// TIA Portal V16 export
// export: Created 2021-04-11T09:51:25.5675002Z, ExportSetting WithDefaults, DisplayName Totally Integrated Automation Portal, DisplayVersion V16, DisplayName TIA Portal Version Control Interface, DisplayVersion V16, DisplayName TIA Portal Openness, DisplayVersion V16, DisplayName STEP 7 Professional, DisplayVersion V16, DisplayName STEP 7 Safety, DisplayVersion V16, DisplayName WinCC Unified SCADA Engineering System, DisplayVersion V16
FUNCTION "DBtoIO" : Void   // FC2, LAD
{ S7_Optimized_Access := 'TRUE' }
VERSION : 0.1
// stored: AutoNumber true, IsIECCheckEnabled false, SetENOAutomatically false, UDAEnableTagReadback false
BEGIN

REGION Network 1: Конвейер1 - вперед
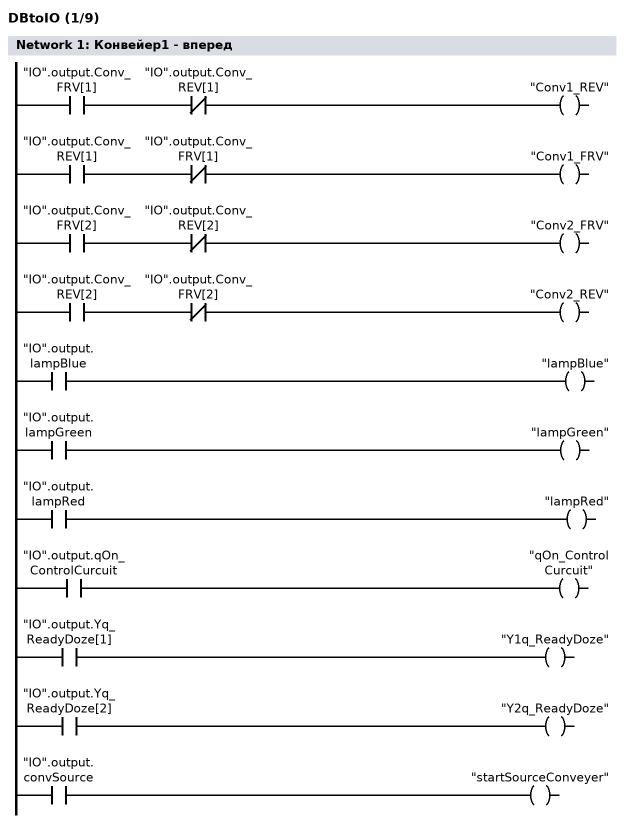
   RUNG wire#powerrail
      Contact( "IO".output.Conv_FRV[1] )
      I_Contact( "IO".output.Conv_REV[1] )
      Coil( "Conv1_REV" )
   END_RUNG
   RUNG wire#powerrail
      Contact( "IO".output.Conv_REV[1] )
      I_Contact( "IO".output.Conv_FRV[1] )
      Coil( "Conv1_FRV" )
   END_RUNG
   RUNG wire#powerrail
      Contact( "IO".output.Conv_FRV[2] )
      I_Contact( "IO".output.Conv_REV[2] )
      Coil( "Conv2_FRV" )
   END_RUNG
   RUNG wire#powerrail
      Contact( "IO".output.Conv_REV[2] )
      I_Contact( "IO".output.Conv_FRV[2] )
      Coil( "Conv2_REV" )
   END_RUNG
   RUNG wire#powerrail
      Contact( "IO".output.lampBlue )
      Coil( "lampBlue" )
   END_RUNG
   RUNG wire#powerrail
      Contact( "IO".output.lampGreen )
      Coil( "lampGreen" )
   END_RUNG
   RUNG wire#powerrail
      Contact( "IO".output.lampRed )
      Coil( "lampRed" )
   END_RUNG
   RUNG wire#powerrail
      Contact( "IO".output.qOn_ControlCurcuit )
      Coil( "qOn_ControlCurcuit" )
   END_RUNG
   RUNG wire#powerrail
      Contact( "IO".output.Yq_ReadyDoze[1] )
      Coil( "Y1q_ReadyDoze" )
   END_RUNG
   RUNG wire#powerrail
      Contact( "IO".output.Yq_ReadyDoze[2] )
      Coil( "Y2q_ReadyDoze" )
   END_RUNG
   RUNG wire#powerrail
      Contact( "IO".output.convSource )
      Coil( "startSourceConveyer" )
   END_RUNG
   // the same network as SCL:
   "Conv1_REV" := "IO".output.Conv_FRV[1] AND NOT "IO".output.Conv_REV[1];
   "Conv1_FRV" := "IO".output.Conv_REV[1] AND NOT "IO".output.Conv_FRV[1];
   "Conv2_FRV" := "IO".output.Conv_FRV[2] AND NOT "IO".output.Conv_REV[2];
   "Conv2_REV" := "IO".output.Conv_REV[2] AND NOT "IO".output.Conv_FRV[2];
   "lampBlue" := "IO".output.lampBlue;
   "lampGreen" := "IO".output.lampGreen;
   "lampRed" := "IO".output.lampRed;
   "qOn_ControlCurcuit" := "IO".output.qOn_ControlCurcuit;
   "Y1q_ReadyDoze" := "IO".output.Yq_ReadyDoze[1];
   "Y2q_ReadyDoze" := "IO".output.Yq_ReadyDoze[2];
   "startSourceConveyer" := "IO".output.convSource;
END_REGION

REGION Network 2: Управление открыванием лопаток - из массива в катушки
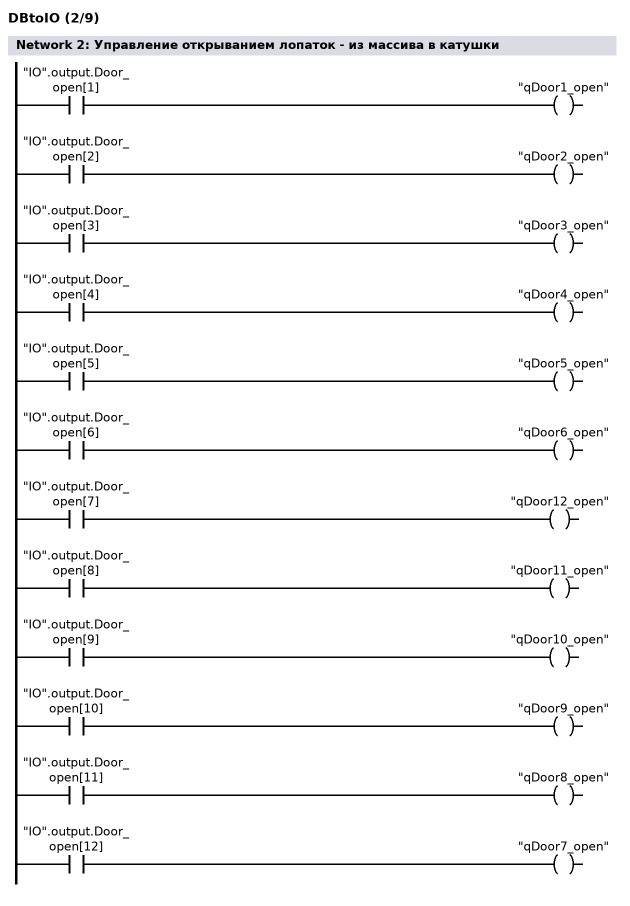
   RUNG wire#powerrail
      Contact( "IO".output.Door_open[1] )
      Coil( "qDoor1_open" )
   END_RUNG
   RUNG wire#powerrail
      Contact( "IO".output.Door_open[2] )
      Coil( "qDoor2_open" )
   END_RUNG
   RUNG wire#powerrail
      Contact( "IO".output.Door_open[3] )
      Coil( "qDoor3_open" )
   END_RUNG
   RUNG wire#powerrail
      Contact( "IO".output.Door_open[4] )
      Coil( "qDoor4_open" )
   END_RUNG
   RUNG wire#powerrail
      Contact( "IO".output.Door_open[5] )
      Coil( "qDoor5_open" )
   END_RUNG
   RUNG wire#powerrail
      Contact( "IO".output.Door_open[6] )
      Coil( "qDoor6_open" )
   END_RUNG
   RUNG wire#powerrail
      Contact( "IO".output.Door_open[7] )
      Coil( "qDoor12_open" )
   END_RUNG
   RUNG wire#powerrail
      Contact( "IO".output.Door_open[8] )
      Coil( "qDoor11_open" )
   END_RUNG
   RUNG wire#powerrail
      Contact( "IO".output.Door_open[9] )
      Coil( "qDoor10_open" )
   END_RUNG
   RUNG wire#powerrail
      Contact( "IO".output.Door_open[10] )
      Coil( "qDoor9_open" )
   END_RUNG
   RUNG wire#powerrail
      Contact( "IO".output.Door_open[11] )
      Coil( "qDoor8_open" )
   END_RUNG
   RUNG wire#powerrail
      Contact( "IO".output.Door_open[12] )
      Coil( "qDoor7_open" )
   END_RUNG
   // the same network as SCL:
   "qDoor1_open" := "IO".output.Door_open[1];
   "qDoor2_open" := "IO".output.Door_open[2];
   "qDoor3_open" := "IO".output.Door_open[3];
   "qDoor4_open" := "IO".output.Door_open[4];
   "qDoor5_open" := "IO".output.Door_open[5];
   "qDoor6_open" := "IO".output.Door_open[6];
   "qDoor12_open" := "IO".output.Door_open[7];
   "qDoor11_open" := "IO".output.Door_open[8];
   "qDoor10_open" := "IO".output.Door_open[9];
   "qDoor9_open" := "IO".output.Door_open[10];
   "qDoor8_open" := "IO".output.Door_open[11];
   "qDoor7_open" := "IO".output.Door_open[12];
END_REGION

REGION Network 3: Управление лопатки закрыть - из массива в катушки
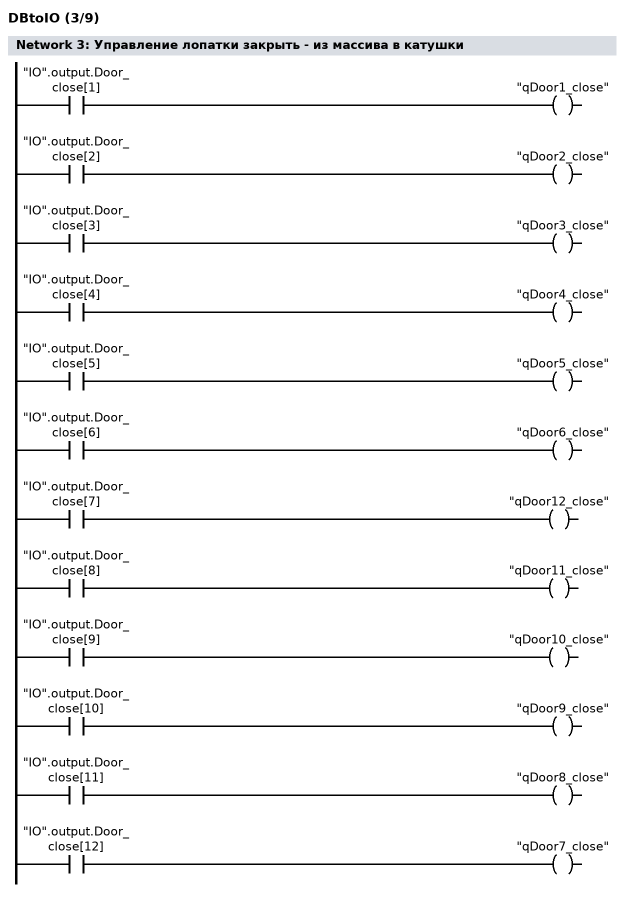
   RUNG wire#powerrail
      Contact( "IO".output.Door_close[1] )
      Coil( "qDoor1_close" )
   END_RUNG
   RUNG wire#powerrail
      Contact( "IO".output.Door_close[2] )
      Coil( "qDoor2_close" )
   END_RUNG
   RUNG wire#powerrail
      Contact( "IO".output.Door_close[3] )
      Coil( "qDoor3_close" )
   END_RUNG
   RUNG wire#powerrail
      Contact( "IO".output.Door_close[4] )
      Coil( "qDoor4_close" )
   END_RUNG
   RUNG wire#powerrail
      Contact( "IO".output.Door_close[5] )
      Coil( "qDoor5_close" )
   END_RUNG
   RUNG wire#powerrail
      Contact( "IO".output.Door_close[6] )
      Coil( "qDoor6_close" )
   END_RUNG
   RUNG wire#powerrail
      Contact( "IO".output.Door_close[7] )
      Coil( "qDoor12_close" )
   END_RUNG
   RUNG wire#powerrail
      Contact( "IO".output.Door_close[8] )
      Coil( "qDoor11_close" )
   END_RUNG
   RUNG wire#powerrail
      Contact( "IO".output.Door_close[9] )
      Coil( "qDoor10_close" )
   END_RUNG
   RUNG wire#powerrail
      Contact( "IO".output.Door_close[10] )
      Coil( "qDoor9_close" )
   END_RUNG
   RUNG wire#powerrail
      Contact( "IO".output.Door_close[11] )
      Coil( "qDoor8_close" )
   END_RUNG
   RUNG wire#powerrail
      Contact( "IO".output.Door_close[12] )
      Coil( "qDoor7_close" )
   END_RUNG
   // the same network as SCL:
   "qDoor1_close" := "IO".output.Door_close[1];
   "qDoor2_close" := "IO".output.Door_close[2];
   "qDoor3_close" := "IO".output.Door_close[3];
   "qDoor4_close" := "IO".output.Door_close[4];
   "qDoor5_close" := "IO".output.Door_close[5];
   "qDoor6_close" := "IO".output.Door_close[6];
   "qDoor12_close" := "IO".output.Door_close[7];
   "qDoor11_close" := "IO".output.Door_close[8];
   "qDoor10_close" := "IO".output.Door_close[9];
   "qDoor9_close" := "IO".output.Door_close[10];
   "qDoor8_close" := "IO".output.Door_close[11];
   "qDoor7_close" := "IO".output.Door_close[12];
END_REGION

REGION Network 4: Управление открыванием левым бункером - из массива в катушки
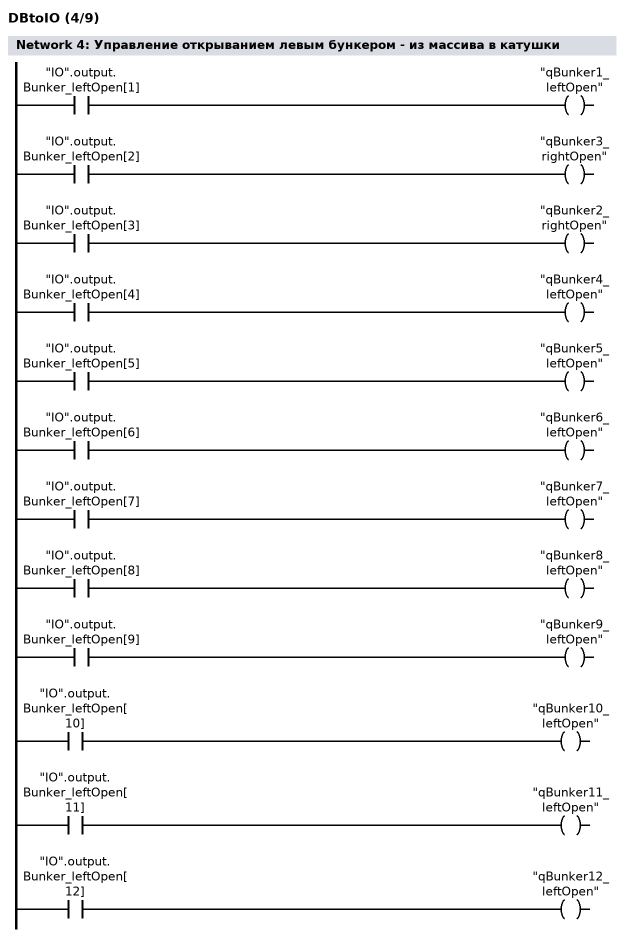
   RUNG wire#powerrail
      Contact( "IO".output.Bunker_leftOpen[1] )
      Coil( "qBunker1_leftOpen" )
   END_RUNG
   RUNG wire#powerrail
      Contact( "IO".output.Bunker_leftOpen[2] )
      Coil( "qBunker3_rightOpen" )
   END_RUNG
   RUNG wire#powerrail
      Contact( "IO".output.Bunker_leftOpen[3] )
      Coil( "qBunker2_rightOpen" )
   END_RUNG
   RUNG wire#powerrail
      Contact( "IO".output.Bunker_leftOpen[4] )
      Coil( "qBunker4_leftOpen" )
   END_RUNG
   RUNG wire#powerrail
      Contact( "IO".output.Bunker_leftOpen[5] )
      Coil( "qBunker5_leftOpen" )
   END_RUNG
   RUNG wire#powerrail
      Contact( "IO".output.Bunker_leftOpen[6] )
      Coil( "qBunker6_leftOpen" )
   END_RUNG
   RUNG wire#powerrail
      Contact( "IO".output.Bunker_leftOpen[7] )
      Coil( "qBunker7_leftOpen" )
   END_RUNG
   RUNG wire#powerrail
      Contact( "IO".output.Bunker_leftOpen[8] )
      Coil( "qBunker8_leftOpen" )
   END_RUNG
   RUNG wire#powerrail
      Contact( "IO".output.Bunker_leftOpen[9] )
      Coil( "qBunker9_leftOpen" )
   END_RUNG
   RUNG wire#powerrail
      Contact( "IO".output.Bunker_leftOpen[10] )
      Coil( "qBunker10_leftOpen" )
   END_RUNG
   RUNG wire#powerrail
      Contact( "IO".output.Bunker_leftOpen[11] )
      Coil( "qBunker11_leftOpen" )
   END_RUNG
   RUNG wire#powerrail
      Contact( "IO".output.Bunker_leftOpen[12] )
      Coil( "qBunker12_leftOpen" )
   END_RUNG
   // the same network as SCL:
   "qBunker1_leftOpen" := "IO".output.Bunker_leftOpen[1];
   "qBunker3_rightOpen" := "IO".output.Bunker_leftOpen[2];
   "qBunker2_rightOpen" := "IO".output.Bunker_leftOpen[3];
   "qBunker4_leftOpen" := "IO".output.Bunker_leftOpen[4];
   "qBunker5_leftOpen" := "IO".output.Bunker_leftOpen[5];
   "qBunker6_leftOpen" := "IO".output.Bunker_leftOpen[6];
   "qBunker7_leftOpen" := "IO".output.Bunker_leftOpen[7];
   "qBunker8_leftOpen" := "IO".output.Bunker_leftOpen[8];
   "qBunker9_leftOpen" := "IO".output.Bunker_leftOpen[9];
   "qBunker10_leftOpen" := "IO".output.Bunker_leftOpen[10];
   "qBunker11_leftOpen" := "IO".output.Bunker_leftOpen[11];
   "qBunker12_leftOpen" := "IO".output.Bunker_leftOpen[12];
END_REGION

REGION Network 5: Управление закрытием левым бункером - из массива в катушки
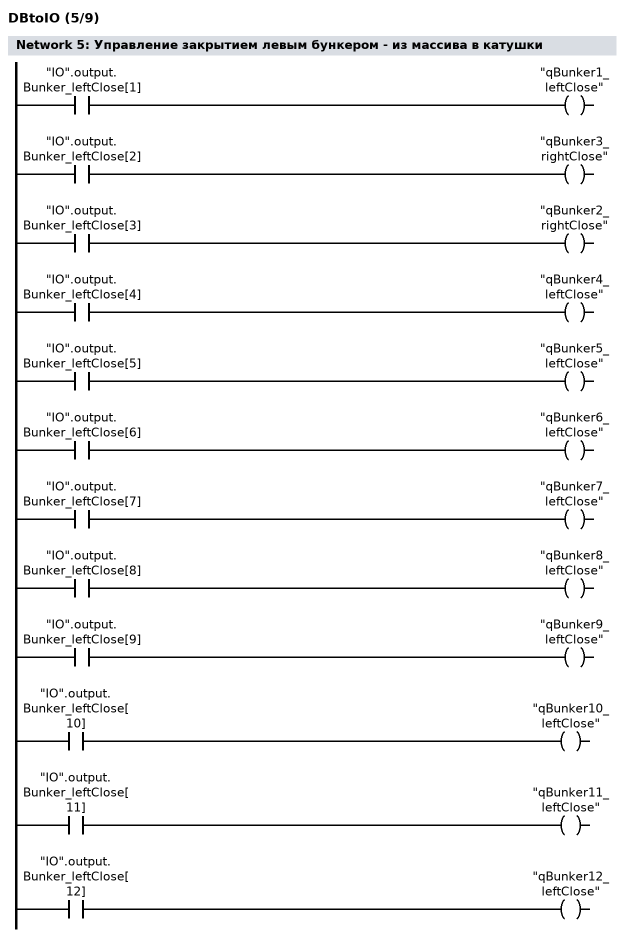
   RUNG wire#powerrail
      Contact( "IO".output.Bunker_leftClose[1] )
      Coil( "qBunker1_leftClose" )
   END_RUNG
   RUNG wire#powerrail
      Contact( "IO".output.Bunker_leftClose[2] )
      Coil( "qBunker3_rightClose" )
   END_RUNG
   RUNG wire#powerrail
      Contact( "IO".output.Bunker_leftClose[3] )
      Coil( "qBunker2_rightClose" )
   END_RUNG
   RUNG wire#powerrail
      Contact( "IO".output.Bunker_leftClose[4] )
      Coil( "qBunker4_leftClose" )
   END_RUNG
   RUNG wire#powerrail
      Contact( "IO".output.Bunker_leftClose[5] )
      Coil( "qBunker5_leftClose" )
   END_RUNG
   RUNG wire#powerrail
      Contact( "IO".output.Bunker_leftClose[6] )
      Coil( "qBunker6_leftClose" )
   END_RUNG
   RUNG wire#powerrail
      Contact( "IO".output.Bunker_leftClose[7] )
      Coil( "qBunker7_leftClose" )
   END_RUNG
   RUNG wire#powerrail
      Contact( "IO".output.Bunker_leftClose[8] )
      Coil( "qBunker8_leftClose" )
   END_RUNG
   RUNG wire#powerrail
      Contact( "IO".output.Bunker_leftClose[9] )
      Coil( "qBunker9_leftClose" )
   END_RUNG
   RUNG wire#powerrail
      Contact( "IO".output.Bunker_leftClose[10] )
      Coil( "qBunker10_leftClose" )
   END_RUNG
   RUNG wire#powerrail
      Contact( "IO".output.Bunker_leftClose[11] )
      Coil( "qBunker11_leftClose" )
   END_RUNG
   RUNG wire#powerrail
      Contact( "IO".output.Bunker_leftClose[12] )
      Coil( "qBunker12_leftClose" )
   END_RUNG
   // the same network as SCL:
   "qBunker1_leftClose" := "IO".output.Bunker_leftClose[1];
   "qBunker3_rightClose" := "IO".output.Bunker_leftClose[2];
   "qBunker2_rightClose" := "IO".output.Bunker_leftClose[3];
   "qBunker4_leftClose" := "IO".output.Bunker_leftClose[4];
   "qBunker5_leftClose" := "IO".output.Bunker_leftClose[5];
   "qBunker6_leftClose" := "IO".output.Bunker_leftClose[6];
   "qBunker7_leftClose" := "IO".output.Bunker_leftClose[7];
   "qBunker8_leftClose" := "IO".output.Bunker_leftClose[8];
   "qBunker9_leftClose" := "IO".output.Bunker_leftClose[9];
   "qBunker10_leftClose" := "IO".output.Bunker_leftClose[10];
   "qBunker11_leftClose" := "IO".output.Bunker_leftClose[11];
   "qBunker12_leftClose" := "IO".output.Bunker_leftClose[12];
END_REGION

REGION Network 6: Управление открыванием правого бункера - из массива в катушки
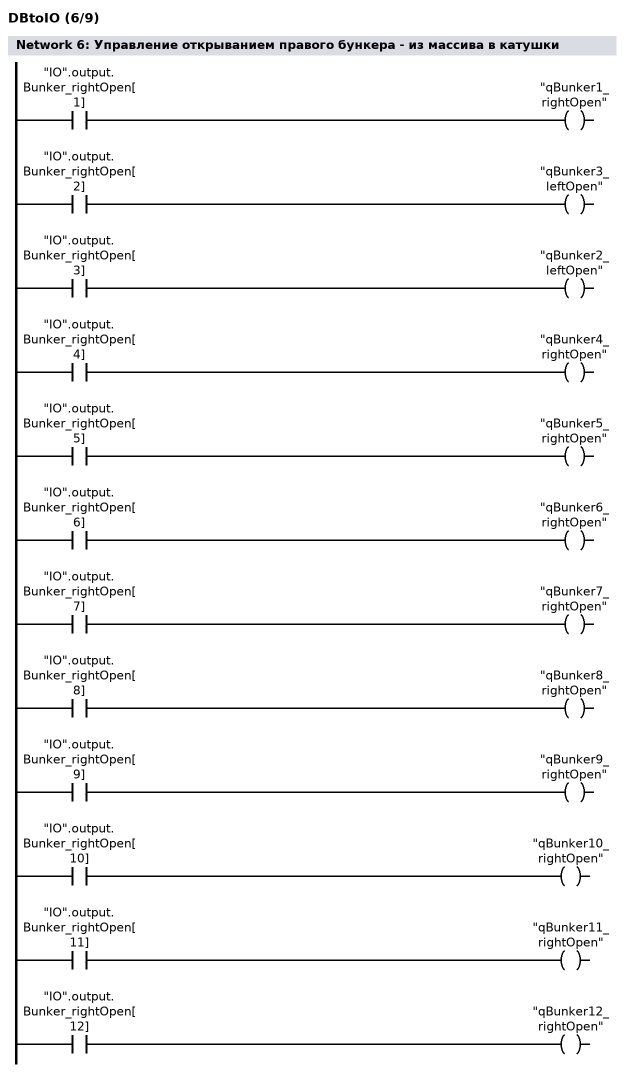
   RUNG wire#powerrail
      Contact( "IO".output.Bunker_rightOpen[1] )
      Coil( "qBunker1_rightOpen" )
   END_RUNG
   RUNG wire#powerrail
      Contact( "IO".output.Bunker_rightOpen[2] )
      Coil( "qBunker3_leftOpen" )
   END_RUNG
   RUNG wire#powerrail
      Contact( "IO".output.Bunker_rightOpen[3] )
      Coil( "qBunker2_leftOpen" )
   END_RUNG
   RUNG wire#powerrail
      Contact( "IO".output.Bunker_rightOpen[4] )
      Coil( "qBunker4_rightOpen" )
   END_RUNG
   RUNG wire#powerrail
      Contact( "IO".output.Bunker_rightOpen[5] )
      Coil( "qBunker5_rightOpen" )
   END_RUNG
   RUNG wire#powerrail
      Contact( "IO".output.Bunker_rightOpen[6] )
      Coil( "qBunker6_rightOpen" )
   END_RUNG
   RUNG wire#powerrail
      Contact( "IO".output.Bunker_rightOpen[7] )
      Coil( "qBunker7_rightOpen" )
   END_RUNG
   RUNG wire#powerrail
      Contact( "IO".output.Bunker_rightOpen[8] )
      Coil( "qBunker8_rightOpen" )
   END_RUNG
   RUNG wire#powerrail
      Contact( "IO".output.Bunker_rightOpen[9] )
      Coil( "qBunker9_rightOpen" )
   END_RUNG
   RUNG wire#powerrail
      Contact( "IO".output.Bunker_rightOpen[10] )
      Coil( "qBunker10_rightOpen" )
   END_RUNG
   RUNG wire#powerrail
      Contact( "IO".output.Bunker_rightOpen[11] )
      Coil( "qBunker11_rightOpen" )
   END_RUNG
   RUNG wire#powerrail
      Contact( "IO".output.Bunker_rightOpen[12] )
      Coil( "qBunker12_rightOpen" )
   END_RUNG
   // the same network as SCL:
   "qBunker1_rightOpen" := "IO".output.Bunker_rightOpen[1];
   "qBunker3_leftOpen" := "IO".output.Bunker_rightOpen[2];
   "qBunker2_leftOpen" := "IO".output.Bunker_rightOpen[3];
   "qBunker4_rightOpen" := "IO".output.Bunker_rightOpen[4];
   "qBunker5_rightOpen" := "IO".output.Bunker_rightOpen[5];
   "qBunker6_rightOpen" := "IO".output.Bunker_rightOpen[6];
   "qBunker7_rightOpen" := "IO".output.Bunker_rightOpen[7];
   "qBunker8_rightOpen" := "IO".output.Bunker_rightOpen[8];
   "qBunker9_rightOpen" := "IO".output.Bunker_rightOpen[9];
   "qBunker10_rightOpen" := "IO".output.Bunker_rightOpen[10];
   "qBunker11_rightOpen" := "IO".output.Bunker_rightOpen[11];
   "qBunker12_rightOpen" := "IO".output.Bunker_rightOpen[12];
END_REGION

REGION Network 7: Управление закрыванием правым бункером - из массива в катушки
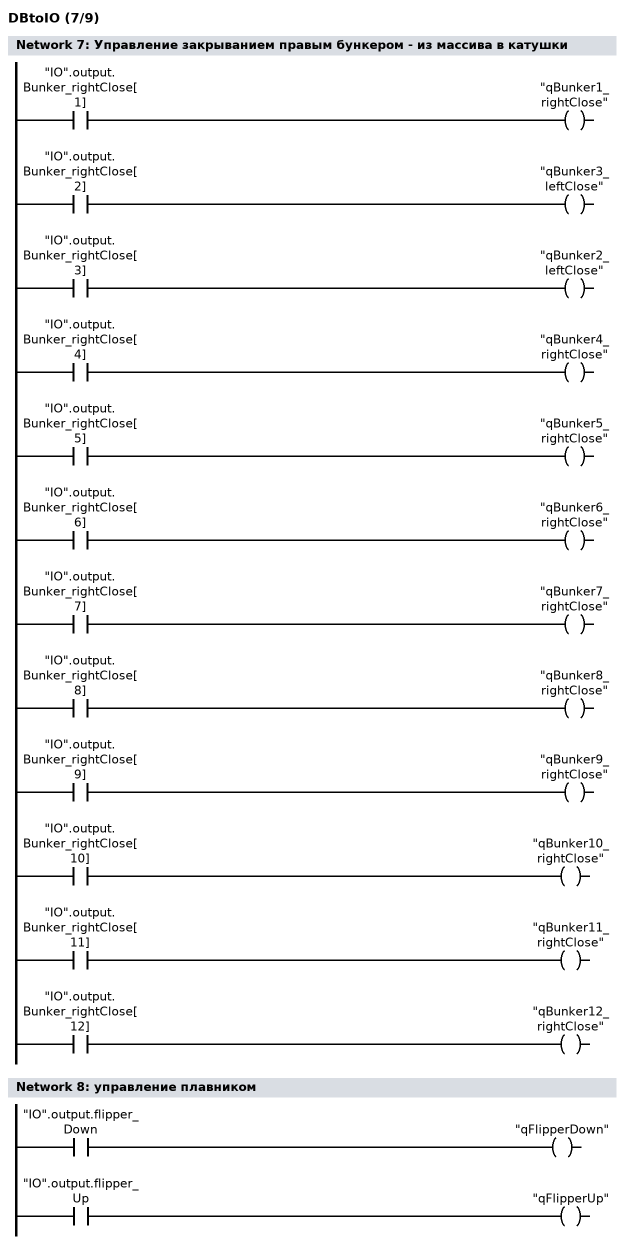
   RUNG wire#powerrail
      Contact( "IO".output.Bunker_rightClose[1] )
      Coil( "qBunker1_rightClose" )
   END_RUNG
   RUNG wire#powerrail
      Contact( "IO".output.Bunker_rightClose[2] )
      Coil( "qBunker3_leftClose" )
   END_RUNG
   RUNG wire#powerrail
      Contact( "IO".output.Bunker_rightClose[3] )
      Coil( "qBunker2_leftClose" )
   END_RUNG
   RUNG wire#powerrail
      Contact( "IO".output.Bunker_rightClose[4] )
      Coil( "qBunker4_rightClose" )
   END_RUNG
   RUNG wire#powerrail
      Contact( "IO".output.Bunker_rightClose[5] )
      Coil( "qBunker5_rightClose" )
   END_RUNG
   RUNG wire#powerrail
      Contact( "IO".output.Bunker_rightClose[6] )
      Coil( "qBunker6_rightClose" )
   END_RUNG
   RUNG wire#powerrail
      Contact( "IO".output.Bunker_rightClose[7] )
      Coil( "qBunker7_rightClose" )
   END_RUNG
   RUNG wire#powerrail
      Contact( "IO".output.Bunker_rightClose[8] )
      Coil( "qBunker8_rightClose" )
   END_RUNG
   RUNG wire#powerrail
      Contact( "IO".output.Bunker_rightClose[9] )
      Coil( "qBunker9_rightClose" )
   END_RUNG
   RUNG wire#powerrail
      Contact( "IO".output.Bunker_rightClose[10] )
      Coil( "qBunker10_rightClose" )
   END_RUNG
   RUNG wire#powerrail
      Contact( "IO".output.Bunker_rightClose[11] )
      Coil( "qBunker11_rightClose" )
   END_RUNG
   RUNG wire#powerrail
      Contact( "IO".output.Bunker_rightClose[12] )
      Coil( "qBunker12_rightClose" )
   END_RUNG
   // the same network as SCL:
   "qBunker1_rightClose" := "IO".output.Bunker_rightClose[1];
   "qBunker3_leftClose" := "IO".output.Bunker_rightClose[2];
   "qBunker2_leftClose" := "IO".output.Bunker_rightClose[3];
   "qBunker4_rightClose" := "IO".output.Bunker_rightClose[4];
   "qBunker5_rightClose" := "IO".output.Bunker_rightClose[5];
   "qBunker6_rightClose" := "IO".output.Bunker_rightClose[6];
   "qBunker7_rightClose" := "IO".output.Bunker_rightClose[7];
   "qBunker8_rightClose" := "IO".output.Bunker_rightClose[8];
   "qBunker9_rightClose" := "IO".output.Bunker_rightClose[9];
   "qBunker10_rightClose" := "IO".output.Bunker_rightClose[10];
   "qBunker11_rightClose" := "IO".output.Bunker_rightClose[11];
   "qBunker12_rightClose" := "IO".output.Bunker_rightClose[12];
END_REGION

REGION Network 8: управление плавником
   RUNG wire#powerrail
      Contact( "IO".output.flipper_Down )
      Coil( "qFlipperDown" )
   END_RUNG
   RUNG wire#powerrail
      Contact( "IO".output.flipper_Up )
      Coil( "qFlipperUp" )
   END_RUNG
   // the same network as SCL:
   "qFlipperDown" := "IO".output.flipper_Down;
   "qFlipperUp" := "IO".output.flipper_Up;
END_REGION

REGION Network 9: Управление вибростолами
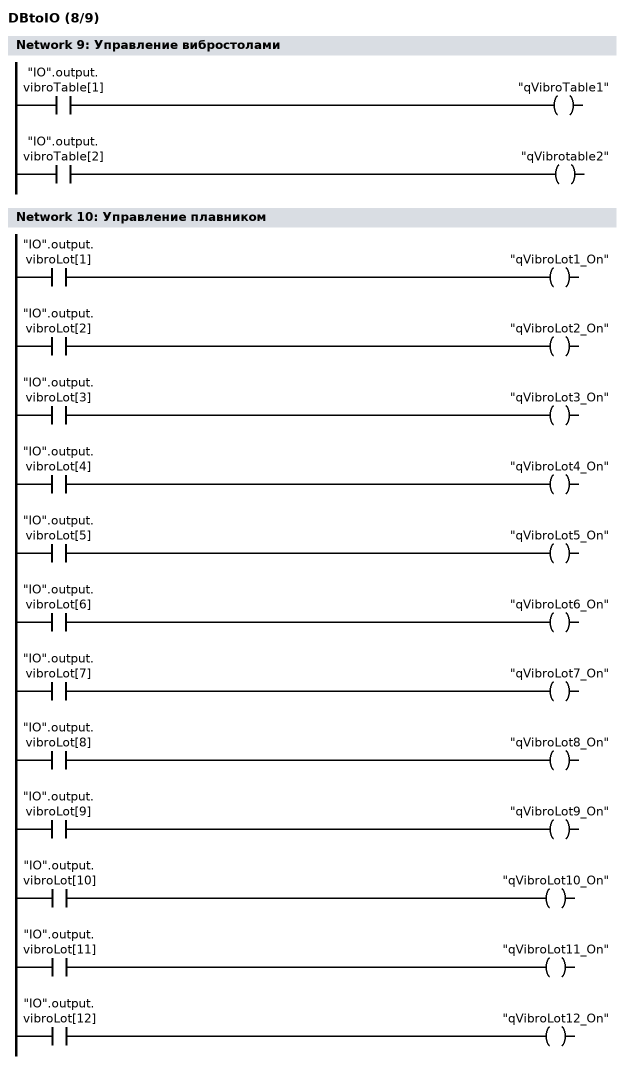
   RUNG wire#powerrail
      Contact( "IO".output.vibroTable[1] )
      Coil( "qVibroTable1" )
   END_RUNG
   RUNG wire#powerrail
      Contact( "IO".output.vibroTable[2] )
      Coil( "qVibrotable2" )
   END_RUNG
   // the same network as SCL:
   "qVibroTable1" := "IO".output.vibroTable[1];
   "qVibrotable2" := "IO".output.vibroTable[2];
END_REGION

REGION Network 10: Управление плавником
   RUNG wire#powerrail
      Contact( "IO".output.vibroLot[1] )
      Coil( "qVibroLot1_On" )
   END_RUNG
   RUNG wire#powerrail
      Contact( "IO".output.vibroLot[2] )
      Coil( "qVibroLot2_On" )
   END_RUNG
   RUNG wire#powerrail
      Contact( "IO".output.vibroLot[3] )
      Coil( "qVibroLot3_On" )
   END_RUNG
   RUNG wire#powerrail
      Contact( "IO".output.vibroLot[4] )
      Coil( "qVibroLot4_On" )
   END_RUNG
   RUNG wire#powerrail
      Contact( "IO".output.vibroLot[5] )
      Coil( "qVibroLot5_On" )
   END_RUNG
   RUNG wire#powerrail
      Contact( "IO".output.vibroLot[6] )
      Coil( "qVibroLot6_On" )
   END_RUNG
   RUNG wire#powerrail
      Contact( "IO".output.vibroLot[7] )
      Coil( "qVibroLot7_On" )
   END_RUNG
   RUNG wire#powerrail
      Contact( "IO".output.vibroLot[8] )
      Coil( "qVibroLot8_On" )
   END_RUNG
   RUNG wire#powerrail
      Contact( "IO".output.vibroLot[9] )
      Coil( "qVibroLot9_On" )
   END_RUNG
   RUNG wire#powerrail
      Contact( "IO".output.vibroLot[10] )
      Coil( "qVibroLot10_On" )
   END_RUNG
   RUNG wire#powerrail
      Contact( "IO".output.vibroLot[11] )
      Coil( "qVibroLot11_On" )
   END_RUNG
   RUNG wire#powerrail
      Contact( "IO".output.vibroLot[12] )
      Coil( "qVibroLot12_On" )
   END_RUNG
   // the same network as SCL:
   "qVibroLot1_On" := "IO".output.vibroLot[1];
   "qVibroLot2_On" := "IO".output.vibroLot[2];
   "qVibroLot3_On" := "IO".output.vibroLot[3];
   "qVibroLot4_On" := "IO".output.vibroLot[4];
   "qVibroLot5_On" := "IO".output.vibroLot[5];
   "qVibroLot6_On" := "IO".output.vibroLot[6];
   "qVibroLot7_On" := "IO".output.vibroLot[7];
   "qVibroLot8_On" := "IO".output.vibroLot[8];
   "qVibroLot9_On" := "IO".output.vibroLot[9];
   "qVibroLot10_On" := "IO".output.vibroLot[10];
   "qVibroLot11_On" := "IO".output.vibroLot[11];
   "qVibroLot12_On" := "IO".output.vibroLot[12];
END_REGION

REGION Network 11: Задание уставки вибрации
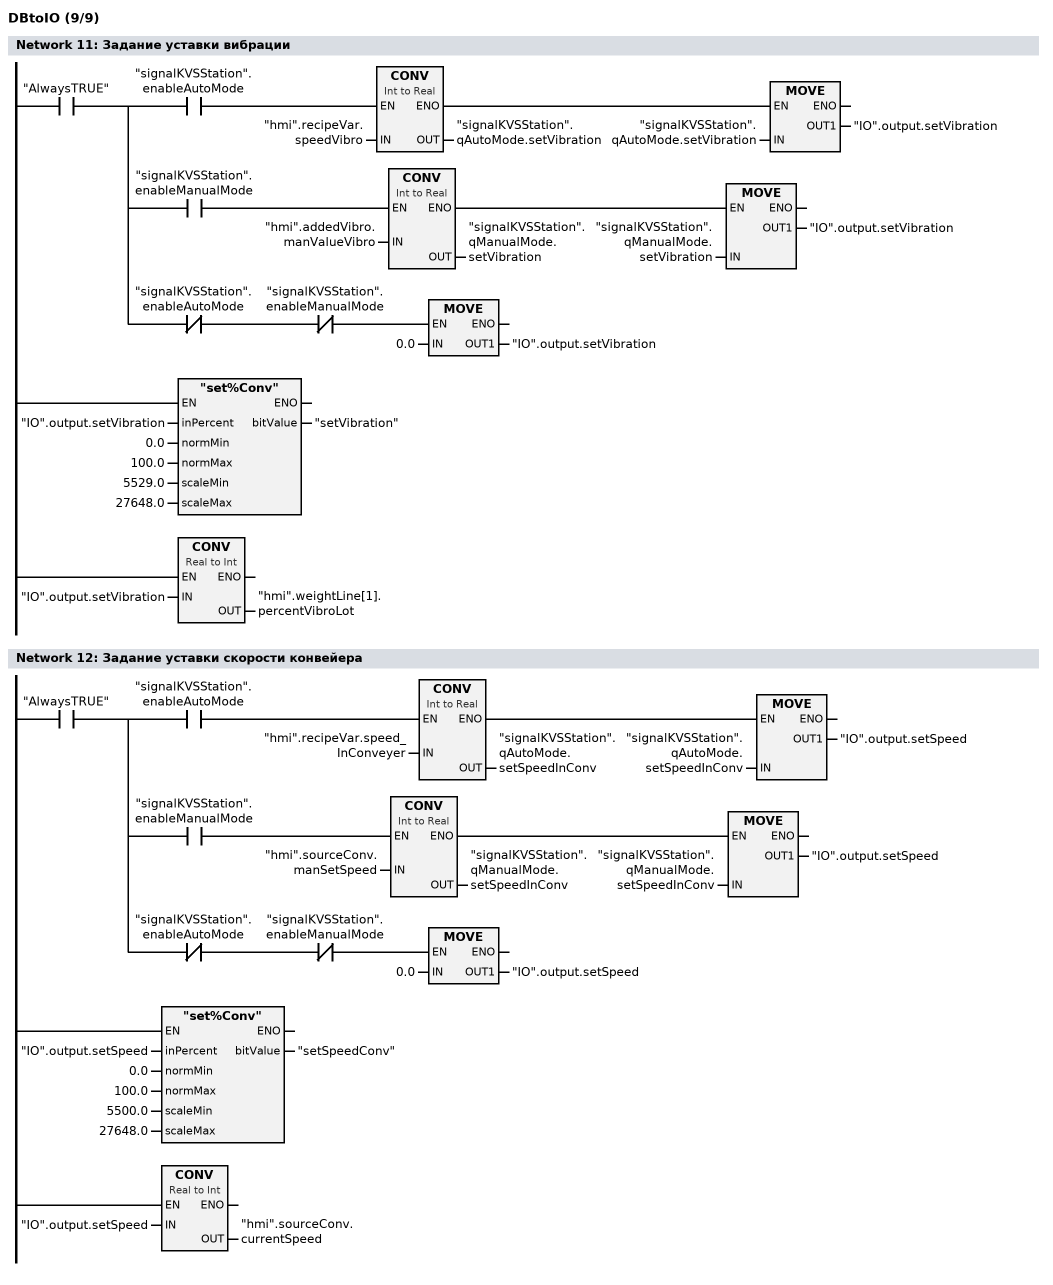
   RUNG wire#powerrail
      Contact( "AlwaysTRUE" )
      wire#w1
      Contact( "signalKVSStation".enableAutoMode )
      { S7_Templates := "[SrcType := Int, DestType := Real]" } Convert(in := "hmi".recipeVar.speedVibro, out => "signalKVSStation".qAutoMode.setVibration)
      Move(in := "signalKVSStation".qAutoMode.setVibration, out1 => "IO".output.setVibration)
   END_RUNG
   RUNG wire#w1
      Contact( "signalKVSStation".enableManualMode )
      { S7_Templates := "[SrcType := Int, DestType := Real]" } Convert(in := "hmi".addedVibro.manValueVibro, out => "signalKVSStation".qManualMode.setVibration)
      Move(in := "signalKVSStation".qManualMode.setVibration, out1 => "IO".output.setVibration)
   END_RUNG
   RUNG wire#w1
      I_Contact( "signalKVSStation".enableAutoMode )
      I_Contact( "signalKVSStation".enableManualMode )
      Move(in := 0.0, out1 => "IO".output.setVibration)
   END_RUNG
   RUNG wire#powerrail
      "set%Conv"(inPercent := "IO".output.setVibration, normMin := 0.0, normMax := 100.0, scaleMin := 5529.0, scaleMax := 27648.0, bitValue => "setVibration")
   END_RUNG
   RUNG wire#powerrail
      { S7_Templates := "[SrcType := Real, DestType := Int]" } Convert(in := "IO".output.setVibration, out => "hmi".weightLine[1].percentVibroLot)
   END_RUNG
   // the same network as SCL:
   IF "AlwaysTRUE" AND "signalKVSStation".enableAutoMode THEN
       "signalKVSStation".qAutoMode.setVibration := INT_TO_REAL("hmi".recipeVar.speedVibro);
       "IO".output.setVibration := "signalKVSStation".qAutoMode.setVibration;
   END_IF;
   IF "AlwaysTRUE" AND "signalKVSStation".enableManualMode THEN
       "signalKVSStation".qManualMode.setVibration := INT_TO_REAL("hmi".addedVibro.manValueVibro);
       "IO".output.setVibration := "signalKVSStation".qManualMode.setVibration;
   END_IF;
   IF "AlwaysTRUE" AND NOT "signalKVSStation".enableAutoMode AND NOT "signalKVSStation".enableManualMode THEN
       "IO".output.setVibration := 0.0;
   END_IF;
   "set%Conv"(inPercent := "IO".output.setVibration,
              normMin := 0.0,
              normMax := 100.0,
              scaleMin := 5529.0,
              scaleMax := 27648.0,
              bitValue => "setVibration");
   "hmi".weightLine[1].percentVibroLot := REAL_TO_INT("IO".output.setVibration);
END_REGION

REGION Network 12: Задание уставки скорости конвейера
   RUNG wire#powerrail
      Contact( "AlwaysTRUE" )
      wire#w1
      Contact( "signalKVSStation".enableAutoMode )
      { S7_Templates := "[SrcType := Int, DestType := Real]" } Convert(in := "hmi".recipeVar.speed_InConveyer, out => "signalKVSStation".qAutoMode.setSpeedInConv)
      Move(in := "signalKVSStation".qAutoMode.setSpeedInConv, out1 => "IO".output.setSpeed)
   END_RUNG
   RUNG wire#w1
      Contact( "signalKVSStation".enableManualMode )
      { S7_Templates := "[SrcType := Int, DestType := Real]" } Convert(in := "hmi".sourceConv.manSetSpeed, out => "signalKVSStation".qManualMode.setSpeedInConv)
      Move(in := "signalKVSStation".qManualMode.setSpeedInConv, out1 => "IO".output.setSpeed)
   END_RUNG
   RUNG wire#w1
      I_Contact( "signalKVSStation".enableAutoMode )
      I_Contact( "signalKVSStation".enableManualMode )
      Move(in := 0.0, out1 => "IO".output.setSpeed)
   END_RUNG
   RUNG wire#powerrail
      "set%Conv"(inPercent := "IO".output.setSpeed, normMin := 0.0, normMax := 100.0, scaleMin := 5500.0, scaleMax := 27648.0, bitValue => "setSpeedConv")
   END_RUNG
   RUNG wire#powerrail
      { S7_Templates := "[SrcType := Real, DestType := Int]" } Convert(in := "IO".output.setSpeed, out => "hmi".sourceConv.currentSpeed)
   END_RUNG
   // the same network as SCL:
   IF "AlwaysTRUE" AND "signalKVSStation".enableAutoMode THEN
       "signalKVSStation".qAutoMode.setSpeedInConv := INT_TO_REAL("hmi".recipeVar.speed_InConveyer);
       "IO".output.setSpeed := "signalKVSStation".qAutoMode.setSpeedInConv;
   END_IF;
   IF "AlwaysTRUE" AND "signalKVSStation".enableManualMode THEN
       "signalKVSStation".qManualMode.setSpeedInConv := INT_TO_REAL("hmi".sourceConv.manSetSpeed);
       "IO".output.setSpeed := "signalKVSStation".qManualMode.setSpeedInConv;
   END_IF;
   IF "AlwaysTRUE" AND NOT "signalKVSStation".enableAutoMode AND NOT "signalKVSStation".enableManualMode THEN
       "IO".output.setSpeed := 0.0;
   END_IF;
   "set%Conv"(inPercent := "IO".output.setSpeed,
              normMin := 0.0,
              normMax := 100.0,
              scaleMin := 5500.0,
              scaleMax := 27648.0,
              bitValue => "setSpeedConv");
   "hmi".sourceConv.currentSpeed := REAL_TO_INT("IO".output.setSpeed);
END_REGION
END_FUNCTION
